VAR_GLOBAL
	var01		:	INT;
END_VAR

(* stored: Version 1.1.0.1, ProductVersion 3.1.4020.6
   GVL GVL01: Id {65ebaf1b-ea2d-45bd-8615-e147f14c91a4} *)
